// Mitsubishi GX Developer project: パレット移載装置   PLC: Q02

PROGRAM T-PANEL
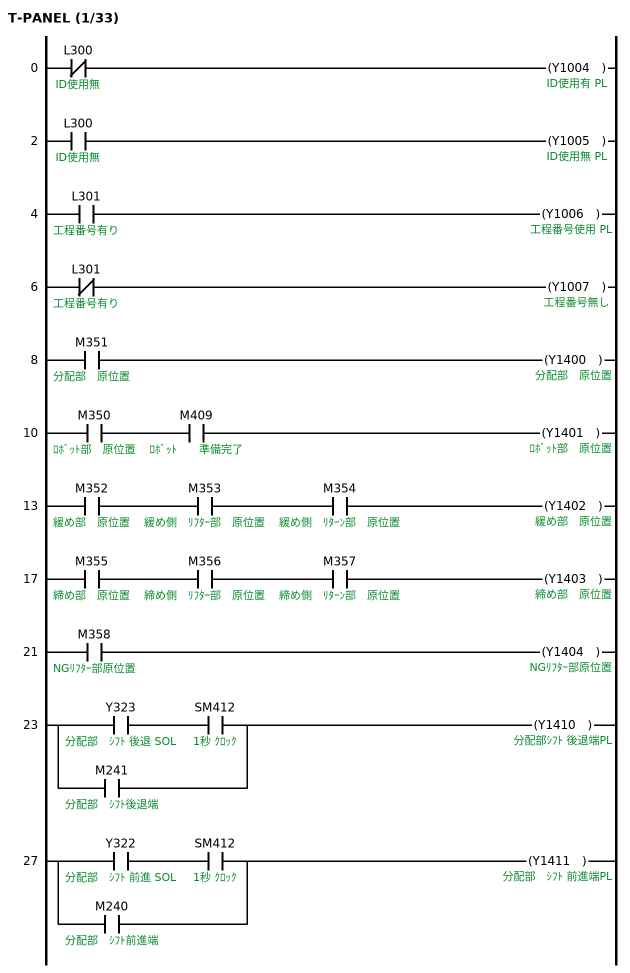
0     LDI     L300  ; ID使用無
      OUT     Y1004  ; ID使用有 PL
2     LD      L300  ; ID使用無
      OUT     Y1005  ; ID使用無 PL
4     LD      L301  ; 工程番号有り
      OUT     Y1006  ; 工程番号使用 PL
6     LDI     L301  ; 工程番号有り
      OUT     Y1007  ; 工程番号無し
8     LD      M351  ; 分配部　原位置
      OUT     Y1400  ; 分配部　原位置
10    LD      M350  ; ﾛﾎﾞｯﾄ部　原位置
      AND     M409  ; ﾛﾎﾞｯﾄ　　準備完了
      OUT     Y1401  ; ﾛﾎﾞｯﾄ部　原位置
13    LD      M352  ; 緩め部　原位置
      AND     M353  ; 緩め側　ﾘﾌﾀｰ部　原位置
      AND     M354  ; 緩め側　ﾘﾀｰﾝ部　原位置
      OUT     Y1402  ; 緩め部　原位置
17    LD      M355  ; 締め部　原位置
      AND     M356  ; 締め側　ﾘﾌﾀｰ部　原位置
      AND     M357  ; 締め側　ﾘﾀｰﾝ部　原位置
      OUT     Y1403  ; 締め部　原位置
21    LD      M358  ; NGﾘﾌﾀｰ部原位置
      OUT     Y1404  ; NGﾘﾌﾀｰ部原位置
23    LD      Y323  ; 分配部　ｼﾌﾄ 後退 SOL
      AND     SM412  ; 1秒 ｸﾛｯｸ
      OR      M241  ; 分配部　ｼﾌﾄ後退端
      OUT     Y1410  ; 分配部ｼﾌﾄ 後退端PL
27    LD      Y322  ; 分配部　ｼﾌﾄ 前進 SOL
      AND     SM412  ; 1秒 ｸﾛｯｸ
      OR      M240  ; 分配部　ｼﾌﾄ前進端
      OUT     Y1411  ; 分配部　ｼﾌﾄ 前進端PL
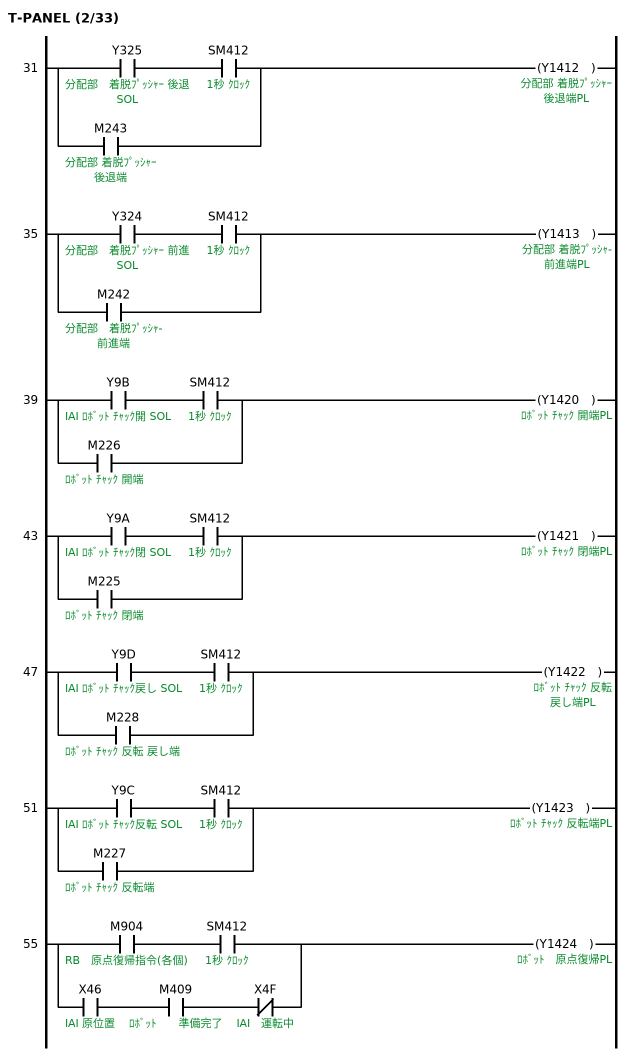
31    LD      Y325  ; 分配部　着脱ﾌﾟｯｼｬｰ 後退 SOL
      AND     SM412  ; 1秒 ｸﾛｯｸ
      OR      M243  ; 分配部 着脱ﾌﾟｯｼｬｰ 後退端
      OUT     Y1412  ; 分配部 着脱ﾌﾟｯｼｬｰ 後退端PL
35    LD      Y324  ; 分配部　着脱ﾌﾟｯｼｬｰ 前進 SOL
      AND     SM412  ; 1秒 ｸﾛｯｸ
      OR      M242  ; 分配部　着脱ﾌﾟｯｼｬ- 前進端
      OUT     Y1413  ; 分配部 着脱ﾌﾟｯｼｬ- 前進端PL
39    LD      Y9B  ; IAI ﾛﾎﾞｯﾄ ﾁｬｯｸ開 SOL
      AND     SM412  ; 1秒 ｸﾛｯｸ
      OR      M226  ; ﾛﾎﾞｯﾄ ﾁｬｯｸ 開端
      OUT     Y1420  ; ﾛﾎﾞｯﾄ ﾁｬｯｸ 開端PL
43    LD      Y9A  ; IAI ﾛﾎﾞｯﾄ ﾁｬｯｸ閉 SOL
      AND     SM412  ; 1秒 ｸﾛｯｸ
      OR      M225  ; ﾛﾎﾞｯﾄ ﾁｬｯｸ 閉端
      OUT     Y1421  ; ﾛﾎﾞｯﾄ ﾁｬｯｸ 閉端PL
47    LD      Y9D  ; IAI ﾛﾎﾞｯﾄ ﾁｬｯｸ戻し SOL
      AND     SM412  ; 1秒 ｸﾛｯｸ
      OR      M228  ; ﾛﾎﾞｯﾄ ﾁｬｯｸ 反転 戻し端
      OUT     Y1422  ; ﾛﾎﾞｯﾄ ﾁｬｯｸ 反転 戻し端PL
51    LD      Y9C  ; IAI ﾛﾎﾞｯﾄ ﾁｬｯｸ反転 SOL
      AND     SM412  ; 1秒 ｸﾛｯｸ
      OR      M227  ; ﾛﾎﾞｯﾄ ﾁｬｯｸ 反転端
      OUT     Y1423  ; ﾛﾎﾞｯﾄ ﾁｬｯｸ 反転端PL
55    LD      M904  ; RB　原点復帰指令(各個)
      AND     SM412  ; 1秒 ｸﾛｯｸ
      LD      X46  ; IAI 原位置
      AND     M409  ; ﾛﾎﾞｯﾄ　　準備完了
      ANI     X4F  ; IAI　運転中
      ORB
      OUT     Y1424  ; ﾛﾎﾞｯﾄ　原点復帰PL
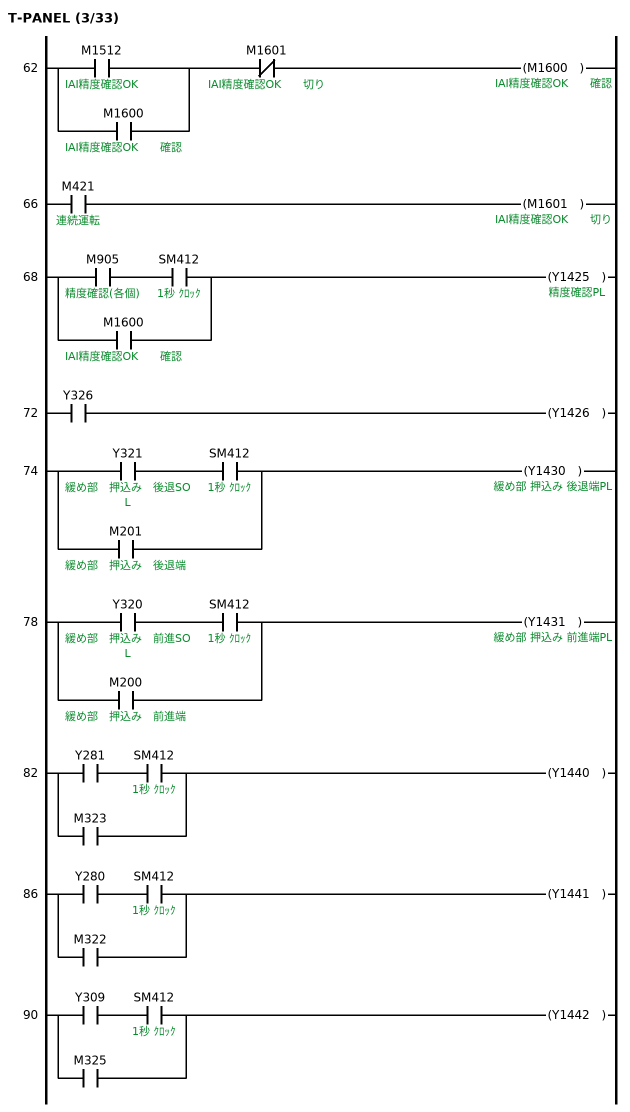
62    LD      M1512  ; IAI精度確認OK
      OR      M1600  ; IAI精度確認OK　　確認
      ANI     M1601  ; IAI精度確認OK　　切り
      OUT     M1600  ; IAI精度確認OK　　確認
66    LD      M421  ; 連続運転
      OUT     M1601  ; IAI精度確認OK　　切り
68    LD      M905  ; 精度確認(各個)
      AND     SM412  ; 1秒 ｸﾛｯｸ
      OR      M1600  ; IAI精度確認OK　　確認
      OUT     Y1425  ; 精度確認PL
72    LD      Y326
      OUT     Y1426
74    LD      Y321  ; 緩め部　押込み　後退SOL
      AND     SM412  ; 1秒 ｸﾛｯｸ
      OR      M201  ; 緩め部　押込み　後退端
      OUT     Y1430  ; 緩め部 押込み 後退端PL
78    LD      Y320  ; 緩め部　押込み　前進SOL
      AND     SM412  ; 1秒 ｸﾛｯｸ
      OR      M200  ; 緩め部　押込み　前進端
      OUT     Y1431  ; 緩め部 押込み 前進端PL
82    LD      Y281
      AND     SM412  ; 1秒 ｸﾛｯｸ
      OR      M323
      OUT     Y1440
86    LD      Y280
      AND     SM412  ; 1秒 ｸﾛｯｸ
      OR      M322
      OUT     Y1441
90    LD      Y309
      AND     SM412  ; 1秒 ｸﾛｯｸ
      OR      M325
      OUT     Y1442
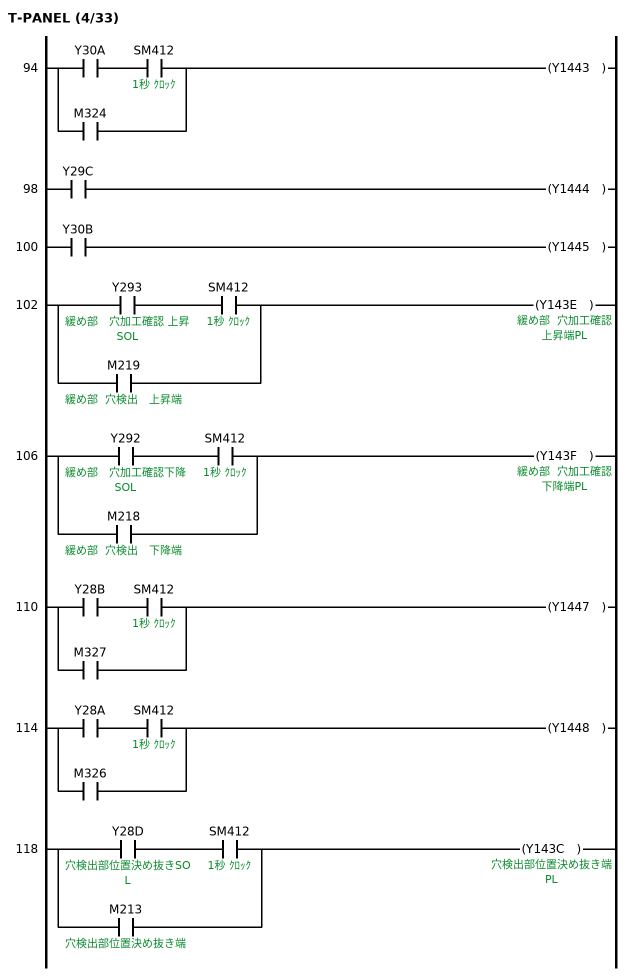
94    LD      Y30A
      AND     SM412  ; 1秒 ｸﾛｯｸ
      OR      M324
      OUT     Y1443
98    LD      Y29C
      OUT     Y1444
100   LD      Y30B
      OUT     Y1445
102   LD      Y293  ; 緩め部　穴加工確認 上昇 SOL
      AND     SM412  ; 1秒 ｸﾛｯｸ
      OR      M219  ; 緩め部  穴検出　上昇端
      OUT     Y143E  ; 緩め部  穴加工確認 上昇端PL
106   LD      Y292  ; 緩め部　穴加工確認下降 SOL
      AND     SM412  ; 1秒 ｸﾛｯｸ
      OR      M218  ; 緩め部  穴検出　下降端
      OUT     Y143F  ; 緩め部  穴加工確認 下降端PL
110   LD      Y28B
      AND     SM412  ; 1秒 ｸﾛｯｸ
      OR      M327
      OUT     Y1447
114   LD      Y28A
      AND     SM412  ; 1秒 ｸﾛｯｸ
      OR      M326
      OUT     Y1448
118   LD      Y28D  ; 穴検出部位置決め抜きSOL
      AND     SM412  ; 1秒 ｸﾛｯｸ
      OR      M213  ; 穴検出部位置決め抜き端
      OUT     Y143C  ; 穴検出部位置決め抜き端PL
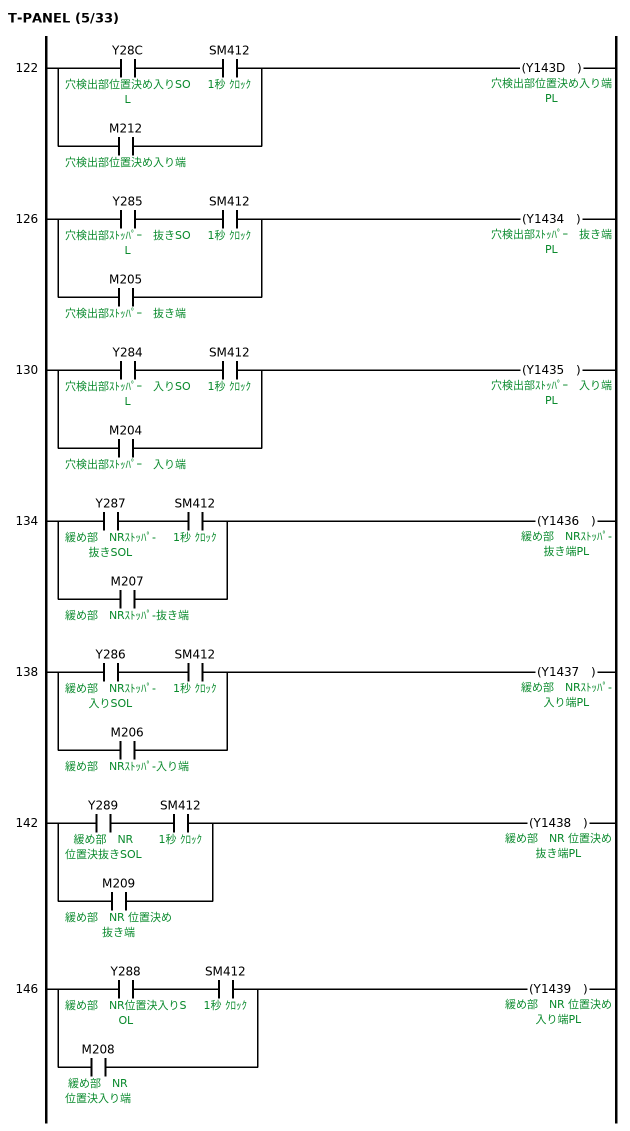
122   LD      Y28C  ; 穴検出部位置決め入りSOL
      AND     SM412  ; 1秒 ｸﾛｯｸ
      OR      M212  ; 穴検出部位置決め入り端
      OUT     Y143D  ; 穴検出部位置決め入り端PL
126   LD      Y285  ; 穴検出部ｽﾄｯﾊﾟｰ　抜きSOL
      AND     SM412  ; 1秒 ｸﾛｯｸ
      OR      M205  ; 穴検出部ｽﾄｯﾊﾟｰ　抜き端
      OUT     Y1434  ; 穴検出部ｽﾄｯﾊﾟｰ　抜き端PL
130   LD      Y284  ; 穴検出部ｽﾄｯﾊﾟｰ　入りSOL
      AND     SM412  ; 1秒 ｸﾛｯｸ
      OR      M204  ; 穴検出部ｽﾄｯﾊﾟｰ　入り端
      OUT     Y1435  ; 穴検出部ｽﾄｯﾊﾟｰ　入り端PL
134   LD      Y287  ; 緩め部　NRｽﾄｯﾊﾟ-抜きSOL
      AND     SM412  ; 1秒 ｸﾛｯｸ
      OR      M207  ; 緩め部　NRｽﾄｯﾊﾟ-抜き端
      OUT     Y1436  ; 緩め部　NRｽﾄｯﾊﾟ-抜き端PL
138   LD      Y286  ; 緩め部　NRｽﾄｯﾊﾟ-入りSOL
      AND     SM412  ; 1秒 ｸﾛｯｸ
      OR      M206  ; 緩め部　NRｽﾄｯﾊﾟ-入り端
      OUT     Y1437  ; 緩め部　NRｽﾄｯﾊﾟ-入り端PL
142   LD      Y289  ; 緩め部　NR 位置決抜きSOL
      AND     SM412  ; 1秒 ｸﾛｯｸ
      OR      M209  ; 緩め部　NR 位置決め 抜き端
      OUT     Y1438  ; 緩め部　NR 位置決め 抜き端PL
146   LD      Y288  ; 緩め部　NR位置決入りSOL
      AND     SM412  ; 1秒 ｸﾛｯｸ
      OR      M208  ; 緩め部　NR 位置決入り端
      OUT     Y1439  ; 緩め部　NR 位置決め 入り端PL
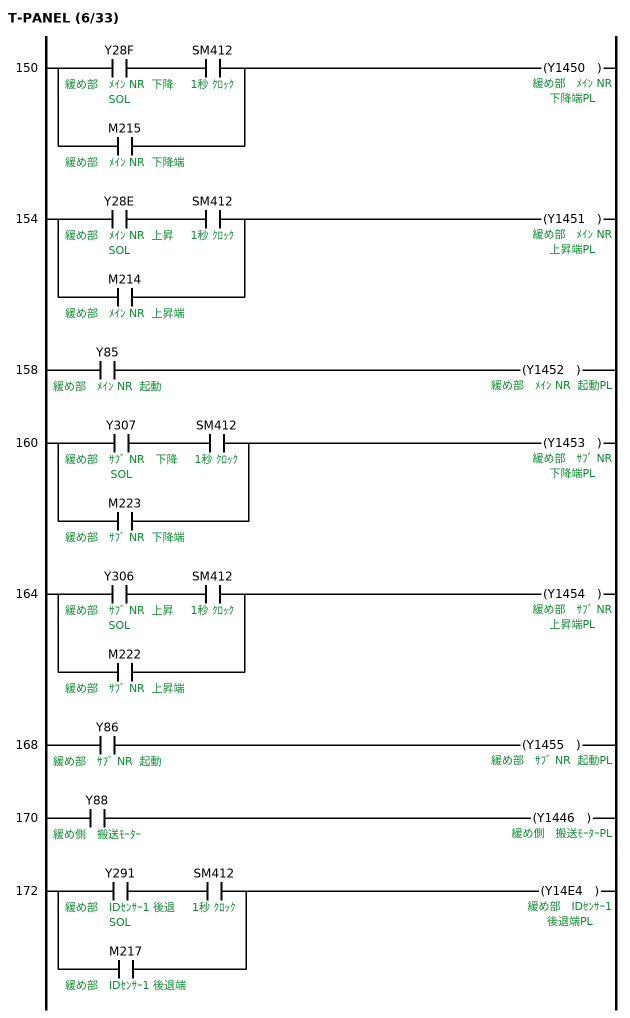
150   LD      Y28F  ; 緩め部　ﾒｲﾝ NR  下降 SOL
      AND     SM412  ; 1秒 ｸﾛｯｸ
      OR      M215  ; 緩め部　ﾒｲﾝ NR  下降端
      OUT     Y1450  ; 緩め部　ﾒｲﾝ NR  下降端PL
154   LD      Y28E  ; 緩め部　ﾒｲﾝ NR  上昇 SOL
      AND     SM412  ; 1秒 ｸﾛｯｸ
      OR      M214  ; 緩め部　ﾒｲﾝ NR  上昇端
      OUT     Y1451  ; 緩め部　ﾒｲﾝ NR  上昇端PL
158   LD      Y85  ; 緩め部　ﾒｲﾝ NR  起動
      OUT     Y1452  ; 緩め部　ﾒｲﾝ NR  起動PL
160   LD      Y307  ; 緩め部　ｻﾌﾞ NR　下降 SOL
      AND     SM412  ; 1秒 ｸﾛｯｸ
      OR      M223  ; 緩め部　ｻﾌﾞ NR  下降端
      OUT     Y1453  ; 緩め部　ｻﾌﾞ NR  下降端PL
164   LD      Y306  ; 緩め部　ｻﾌﾞ NR  上昇 SOL
      AND     SM412  ; 1秒 ｸﾛｯｸ
      OR      M222  ; 緩め部　ｻﾌﾞ NR  上昇端
      OUT     Y1454  ; 緩め部　ｻﾌﾞ NR  上昇端PL
168   LD      Y86  ; 緩め部　ｻﾌﾞ NR  起動
      OUT     Y1455  ; 緩め部　ｻﾌﾞ NR  起動PL
170   LD      Y88  ; 緩め側　搬送ﾓｰﾀｰ
      OUT     Y1446  ; 緩め側　搬送ﾓｰﾀｰPL
172   LD      Y291  ; 緩め部　IDｾﾝｻｰ1 後退 SOL
      AND     SM412  ; 1秒 ｸﾛｯｸ
      OR      M217  ; 緩め部　IDｾﾝｻｰ1 後退端
      OUT     Y14E4  ; 緩め部　IDｾﾝｻｰ1 後退端PL
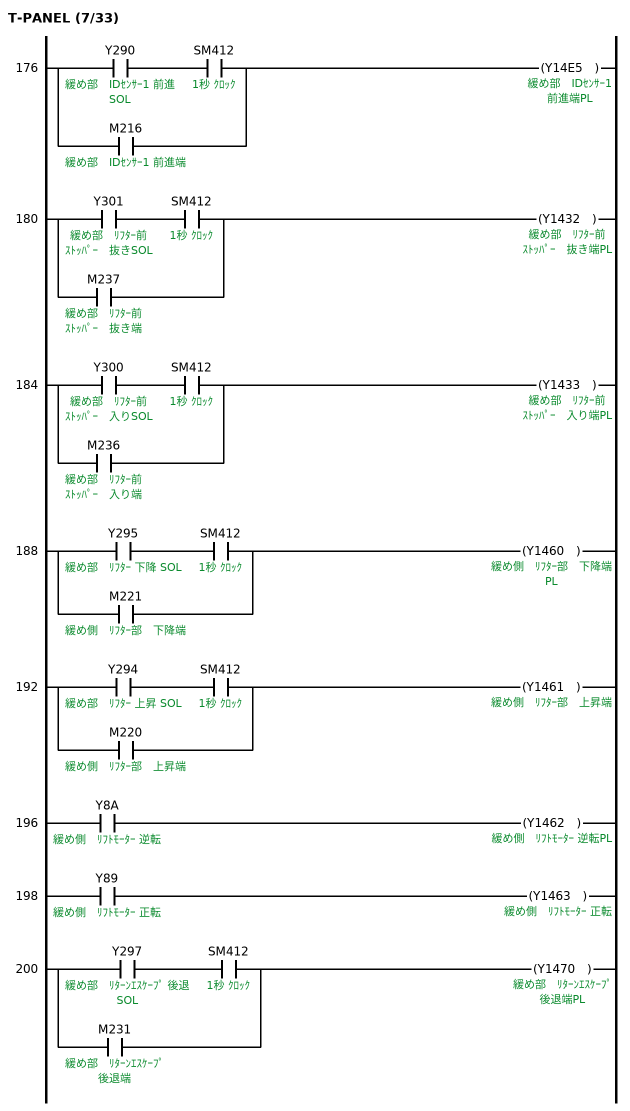
176   LD      Y290  ; 緩め部　IDｾﾝｻｰ1 前進 SOL
      AND     SM412  ; 1秒 ｸﾛｯｸ
      OR      M216  ; 緩め部　IDｾﾝｻｰ1 前進端
      OUT     Y14E5  ; 緩め部　IDｾﾝｻｰ1 前進端PL
180   LD      Y301  ; 緩め部　ﾘﾌﾀｰ前  ｽﾄｯﾊﾟｰ　抜きSOL
      AND     SM412  ; 1秒 ｸﾛｯｸ
      OR      M237  ; 緩め部　ﾘﾌﾀｰ前  ｽﾄｯﾊﾟｰ　抜き端
      OUT     Y1432  ; 緩め部　ﾘﾌﾀｰ前  ｽﾄｯﾊﾟｰ　抜き端PL
184   LD      Y300  ; 緩め部　ﾘﾌﾀｰ前  ｽﾄｯﾊﾟｰ　入りSOL
      AND     SM412  ; 1秒 ｸﾛｯｸ
      OR      M236  ; 緩め部　ﾘﾌﾀｰ前  ｽﾄｯﾊﾟｰ　入り端
      OUT     Y1433  ; 緩め部　ﾘﾌﾀｰ前  ｽﾄｯﾊﾟｰ　入り端PL
188   LD      Y295  ; 緩め部　ﾘﾌﾀｰ 下降 SOL
      AND     SM412  ; 1秒 ｸﾛｯｸ
      OR      M221  ; 緩め側　ﾘﾌﾀｰ部　下降端
      OUT     Y1460  ; 緩め側　ﾘﾌﾀｰ部　下降端PL
192   LD      Y294  ; 緩め部　ﾘﾌﾀｰ 上昇 SOL
      AND     SM412  ; 1秒 ｸﾛｯｸ
      OR      M220  ; 緩め側　ﾘﾌﾀｰ部　上昇端
      OUT     Y1461  ; 緩め側　ﾘﾌﾀｰ部　上昇端
196   LD      Y8A  ; 緩め側　ﾘﾌﾄﾓｰﾀｰ 逆転
      OUT     Y1462  ; 緩め側　ﾘﾌﾄﾓｰﾀｰ 逆転PL
198   LD      Y89  ; 緩め側　ﾘﾌﾄﾓｰﾀｰ 正転
      OUT     Y1463  ; 緩め側　ﾘﾌﾄﾓｰﾀｰ 正転
200   LD      Y297  ; 緩め部　ﾘﾀｰﾝｴｽｹｰﾌﾟ 後退 SOL
      AND     SM412  ; 1秒 ｸﾛｯｸ
      OR      M231  ; 緩め部　ﾘﾀｰﾝｴｽｹｰﾌﾟ 後退端
      OUT     Y1470  ; 緩め部　ﾘﾀｰﾝｴｽｹｰﾌﾟ 後退端PL
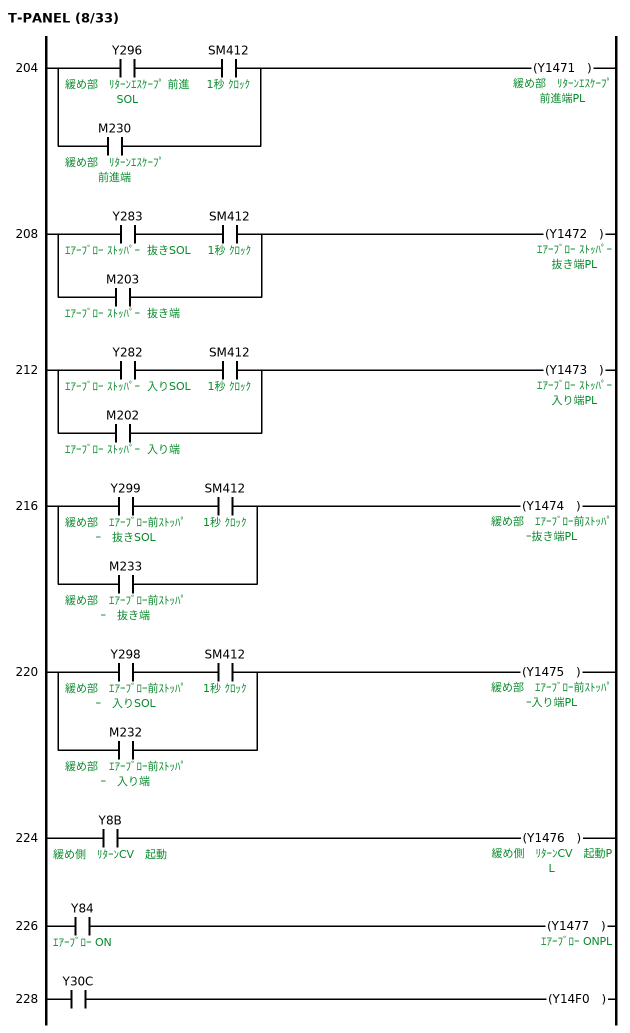
204   LD      Y296  ; 緩め部　ﾘﾀｰﾝｴｽｹｰﾌﾟ 前進 SOL
      AND     SM412  ; 1秒 ｸﾛｯｸ
      OR      M230  ; 緩め部　ﾘﾀｰﾝｴｽｹｰﾌﾟ 前進端
      OUT     Y1471  ; 緩め部　ﾘﾀｰﾝｴｽｹｰﾌﾟ 前進端PL
208   LD      Y283  ; ｴｱｰﾌﾞﾛｰ ｽﾄｯﾊﾟｰ  抜きSOL
      AND     SM412  ; 1秒 ｸﾛｯｸ
      OR      M203  ; ｴｱｰﾌﾞﾛｰ ｽﾄｯﾊﾟｰ  抜き端
      OUT     Y1472  ; ｴｱｰﾌﾞﾛｰ ｽﾄｯﾊﾟｰ  抜き端PL
212   LD      Y282  ; ｴｱｰﾌﾞﾛｰ ｽﾄｯﾊﾟｰ  入りSOL
      AND     SM412  ; 1秒 ｸﾛｯｸ
      OR      M202  ; ｴｱｰﾌﾞﾛｰ ｽﾄｯﾊﾟｰ  入り端
      OUT     Y1473  ; ｴｱｰﾌﾞﾛｰ ｽﾄｯﾊﾟｰ  入り端PL
216   LD      Y299  ; 緩め部　ｴｱｰﾌﾞﾛｰ前ｽﾄｯﾊﾟｰ　抜きSOL
      AND     SM412  ; 1秒 ｸﾛｯｸ
      OR      M233  ; 緩め部　ｴｱｰﾌﾞﾛｰ前ｽﾄｯﾊﾟｰ　抜き端
      OUT     Y1474  ; 緩め部　ｴｱｰﾌﾞﾛｰ前ｽﾄｯﾊﾟｰ抜き端PL
220   LD      Y298  ; 緩め部　ｴｱｰﾌﾞﾛｰ前ｽﾄｯﾊﾟｰ　入りSOL
      AND     SM412  ; 1秒 ｸﾛｯｸ
      OR      M232  ; 緩め部　ｴｱｰﾌﾞﾛｰ前ｽﾄｯﾊﾟｰ　入り端
      OUT     Y1475  ; 緩め部　ｴｱｰﾌﾞﾛｰ前ｽﾄｯﾊﾟｰ入り端PL
224   LD      Y8B  ; 緩め側　ﾘﾀｰﾝCV　起動
      OUT     Y1476  ; 緩め側　ﾘﾀｰﾝCV　起動PL
226   LD      Y84  ; ｴｱｰﾌﾞﾛｰ ON
      OUT     Y1477  ; ｴｱｰﾌﾞﾛｰ ONPL
228   LD      Y30C
      OUT     Y14F0
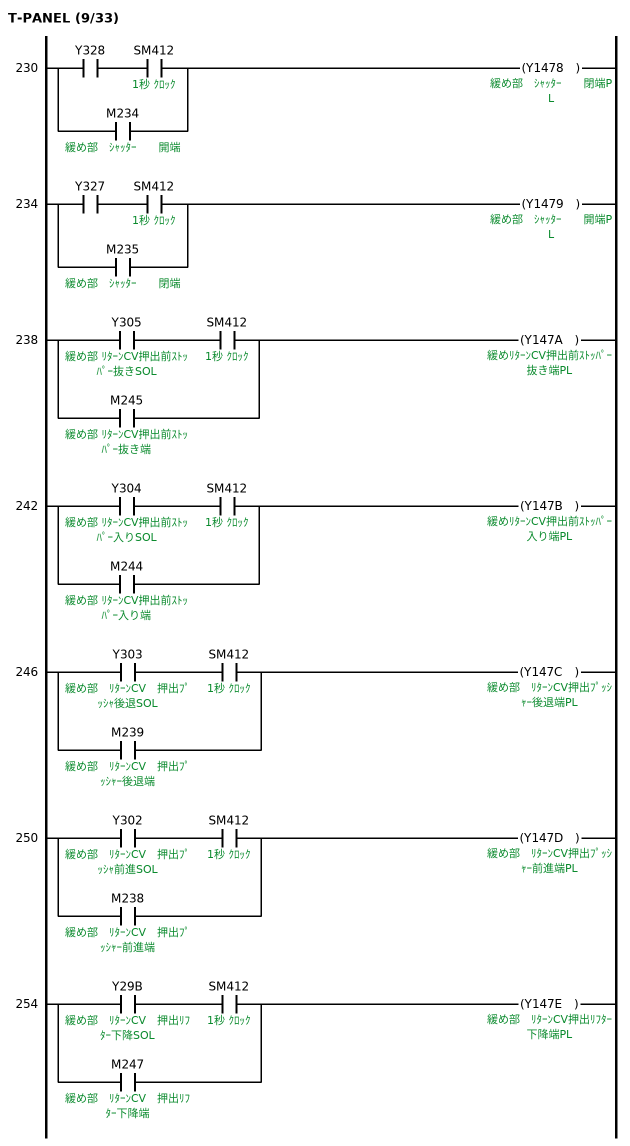
230   LD      Y328
      AND     SM412  ; 1秒 ｸﾛｯｸ
      OR      M234  ; 緩め部　ｼｬｯﾀｰ　　開端
      OUT     Y1478  ; 緩め部　ｼｬｯﾀｰ　　閉端PL
234   LD      Y327
      AND     SM412  ; 1秒 ｸﾛｯｸ
      OR      M235  ; 緩め部　ｼｬｯﾀｰ　　閉端
      OUT     Y1479  ; 緩め部　ｼｬｯﾀｰ　　開端PL
238   LD      Y305  ; 緩め部 ﾘﾀｰﾝCV押出前ｽﾄｯﾊﾟｰ抜きSOL
      AND     SM412  ; 1秒 ｸﾛｯｸ
      OR      M245  ; 緩め部 ﾘﾀｰﾝCV押出前ｽﾄｯﾊﾟｰ抜き端
      OUT     Y147A  ; 緩めﾘﾀｰﾝCV押出前ｽﾄｯﾊﾟｰ抜き端PL
242   LD      Y304  ; 緩め部 ﾘﾀｰﾝCV押出前ｽﾄｯﾊﾟｰ入りSOL
      AND     SM412  ; 1秒 ｸﾛｯｸ
      OR      M244  ; 緩め部 ﾘﾀｰﾝCV押出前ｽﾄｯﾊﾟｰ入り端
      OUT     Y147B  ; 緩めﾘﾀｰﾝCV押出前ｽﾄｯﾊﾟｰ入り端PL
246   LD      Y303  ; 緩め部　ﾘﾀｰﾝCV　押出ﾌﾟｯｼｬ後退SOL
      AND     SM412  ; 1秒 ｸﾛｯｸ
      OR      M239  ; 緩め部　ﾘﾀｰﾝCV　押出ﾌﾟｯｼｬｰ後退端
      OUT     Y147C  ; 緩め部　ﾘﾀｰﾝCV押出ﾌﾟｯｼｬｰ後退端PL
250   LD      Y302  ; 緩め部　ﾘﾀｰﾝCV　押出ﾌﾟｯｼｬ前進SOL
      AND     SM412  ; 1秒 ｸﾛｯｸ
      OR      M238  ; 緩め部　ﾘﾀｰﾝCV　押出ﾌﾟｯｼｬｰ前進端
      OUT     Y147D  ; 緩め部　ﾘﾀｰﾝCV押出ﾌﾟｯｼｬｰ前進端PL
254   LD      Y29B  ; 緩め部　ﾘﾀｰﾝCV　押出ﾘﾌﾀｰ下降SOL
      AND     SM412  ; 1秒 ｸﾛｯｸ
      OR      M247  ; 緩め部　ﾘﾀｰﾝCV　押出ﾘﾌﾀｰ下降端
      OUT     Y147E  ; 緩め部　ﾘﾀｰﾝCV押出ﾘﾌﾀｰ下降端PL
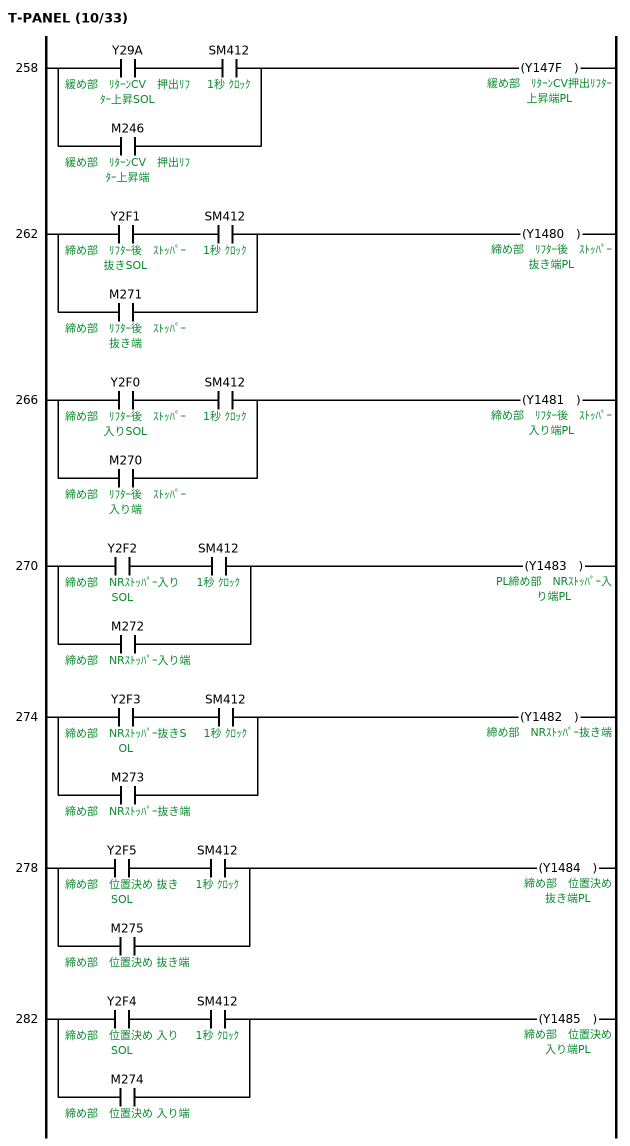
258   LD      Y29A  ; 緩め部　ﾘﾀｰﾝCV　押出ﾘﾌﾀｰ上昇SOL
      AND     SM412  ; 1秒 ｸﾛｯｸ
      OR      M246  ; 緩め部　ﾘﾀｰﾝCV　押出ﾘﾌﾀｰ上昇端
      OUT     Y147F  ; 緩め部　ﾘﾀｰﾝCV押出ﾘﾌﾀｰ上昇端PL
262   LD      Y2F1  ; 締め部　ﾘﾌﾀｰ後　ｽﾄｯﾊﾟｰ　抜きSOL
      AND     SM412  ; 1秒 ｸﾛｯｸ
      OR      M271  ; 締め部　ﾘﾌﾀｰ後　ｽﾄｯﾊﾟｰ　抜き端
      OUT     Y1480  ; 締め部　ﾘﾌﾀｰ後　ｽﾄｯﾊﾟｰ　抜き端PL
266   LD      Y2F0  ; 締め部　ﾘﾌﾀｰ後　ｽﾄｯﾊﾟｰ　入りSOL
      AND     SM412  ; 1秒 ｸﾛｯｸ
      OR      M270  ; 締め部　ﾘﾌﾀｰ後　ｽﾄｯﾊﾟｰ　入り端
      OUT     Y1481  ; 締め部　ﾘﾌﾀｰ後　ｽﾄｯﾊﾟｰ　入り端PL
270   LD      Y2F2  ; 締め部　NRｽﾄｯﾊﾟｰ入り SOL
      AND     SM412  ; 1秒 ｸﾛｯｸ
      OR      M272  ; 締め部　NRｽﾄｯﾊﾟｰ入り端
      OUT     Y1483  ; PL締め部　NRｽﾄｯﾊﾟｰ入り端PL
274   LD      Y2F3  ; 締め部　NRｽﾄｯﾊﾟｰ抜きSOL
      AND     SM412  ; 1秒 ｸﾛｯｸ
      OR      M273  ; 締め部　NRｽﾄｯﾊﾟｰ抜き端
      OUT     Y1482  ; 締め部　NRｽﾄｯﾊﾟｰ抜き端
278   LD      Y2F5  ; 締め部　位置決め 抜き SOL
      AND     SM412  ; 1秒 ｸﾛｯｸ
      OR      M275  ; 締め部　位置決め 抜き端
      OUT     Y1484  ; 締め部　位置決め 抜き端PL
282   LD      Y2F4  ; 締め部　位置決め 入り SOL
      AND     SM412  ; 1秒 ｸﾛｯｸ
      OR      M274  ; 締め部　位置決め 入り端
      OUT     Y1485  ; 締め部　位置決め 入り端PL
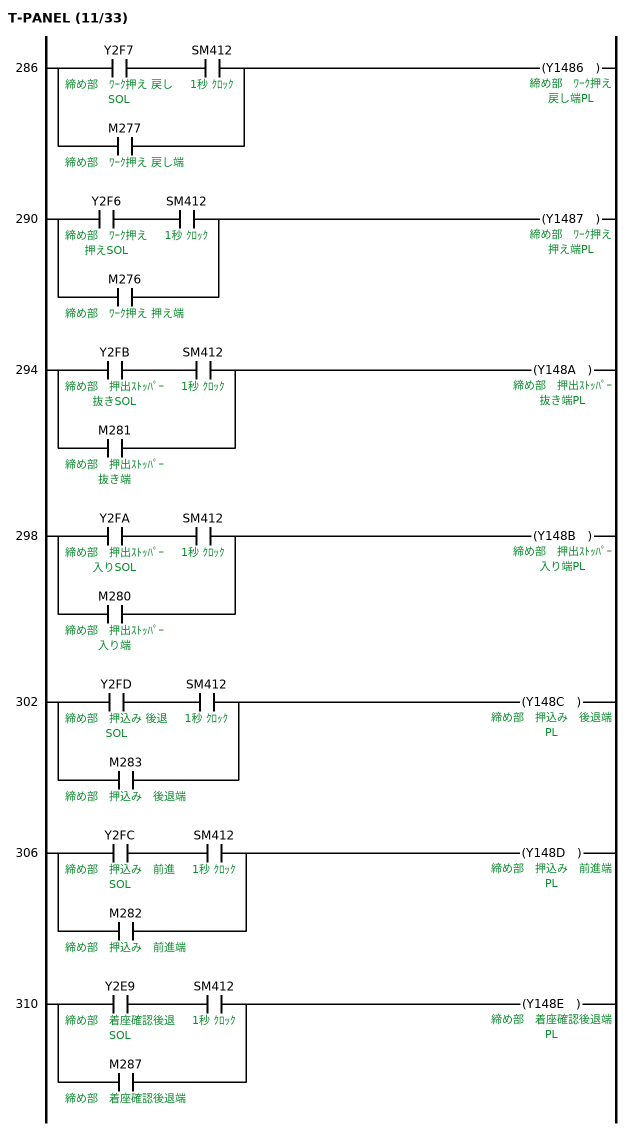
286   LD      Y2F7  ; 締め部　ﾜｰｸ押え 戻し SOL
      AND     SM412  ; 1秒 ｸﾛｯｸ
      OR      M277  ; 締め部　ﾜｰｸ押え 戻し端
      OUT     Y1486  ; 締め部　ﾜｰｸ押え 戻し端PL
290   LD      Y2F6  ; 締め部　ﾜｰｸ押え 押えSOL
      AND     SM412  ; 1秒 ｸﾛｯｸ
      OR      M276  ; 締め部　ﾜｰｸ押え 押え端
      OUT     Y1487  ; 締め部　ﾜｰｸ押え 押え端PL
294   LD      Y2FB  ; 締め部　押出ｽﾄｯﾊﾟｰ 抜きSOL
      AND     SM412  ; 1秒 ｸﾛｯｸ
      OR      M281  ; 締め部　押出ｽﾄｯﾊﾟｰ 抜き端
      OUT     Y148A  ; 締め部　押出ｽﾄｯﾊﾟｰ 抜き端PL
298   LD      Y2FA  ; 締め部　押出ｽﾄｯﾊﾟｰ 入りSOL
      AND     SM412  ; 1秒 ｸﾛｯｸ
      OR      M280  ; 締め部　押出ｽﾄｯﾊﾟｰ 入り端
      OUT     Y148B  ; 締め部　押出ｽﾄｯﾊﾟｰ 入り端PL
302   LD      Y2FD  ; 締め部　押込み 後退 SOL
      AND     SM412  ; 1秒 ｸﾛｯｸ
      OR      M283  ; 締め部　押込み　後退端
      OUT     Y148C  ; 締め部　押込み　後退端PL
306   LD      Y2FC  ; 締め部　押込み　前進 SOL
      AND     SM412  ; 1秒 ｸﾛｯｸ
      OR      M282  ; 締め部　押込み　前進端
      OUT     Y148D  ; 締め部　押込み　前進端PL
310   LD      Y2E9  ; 締め部　着座確認後退 SOL
      AND     SM412  ; 1秒 ｸﾛｯｸ
      OR      M287  ; 締め部　着座確認後退端
      OUT     Y148E  ; 締め部　着座確認後退端PL
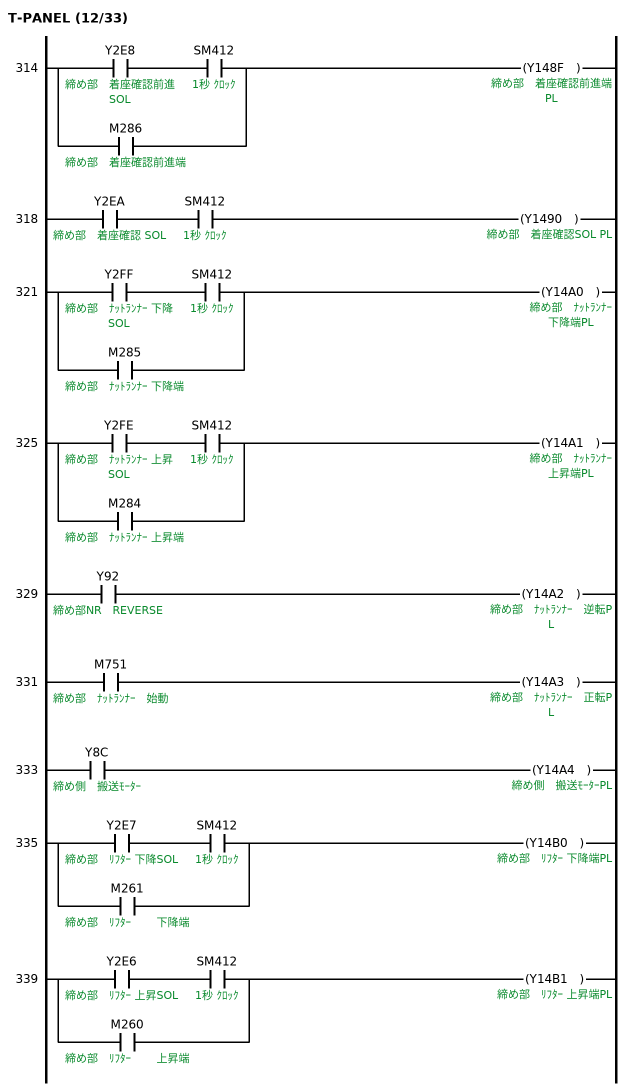
314   LD      Y2E8  ; 締め部　着座確認前進 SOL
      AND     SM412  ; 1秒 ｸﾛｯｸ
      OR      M286  ; 締め部　着座確認前進端
      OUT     Y148F  ; 締め部　着座確認前進端PL
318   LD      Y2EA  ; 締め部　着座確認 SOL
      AND     SM412  ; 1秒 ｸﾛｯｸ
      OUT     Y1490  ; 締め部　着座確認SOL PL
321   LD      Y2FF  ; 締め部　ﾅｯﾄﾗﾝﾅｰ 下降 SOL
      AND     SM412  ; 1秒 ｸﾛｯｸ
      OR      M285  ; 締め部　ﾅｯﾄﾗﾝﾅｰ 下降端
      OUT     Y14A0  ; 締め部　ﾅｯﾄﾗﾝﾅｰ 下降端PL
325   LD      Y2FE  ; 締め部　ﾅｯﾄﾗﾝﾅｰ 上昇 SOL
      AND     SM412  ; 1秒 ｸﾛｯｸ
      OR      M284  ; 締め部　ﾅｯﾄﾗﾝﾅｰ 上昇端
      OUT     Y14A1  ; 締め部　ﾅｯﾄﾗﾝﾅｰ 上昇端PL
329   LD      Y92  ; 締め部NR　REVERSE
      OUT     Y14A2  ; 締め部　ﾅｯﾄﾗﾝﾅｰ　逆転PL
331   LD      M751  ; 締め部　ﾅｯﾄﾗﾝﾅｰ　始動
      OUT     Y14A3  ; 締め部　ﾅｯﾄﾗﾝﾅｰ　正転PL
333   LD      Y8C  ; 締め側　搬送ﾓｰﾀｰ
      OUT     Y14A4  ; 締め側　搬送ﾓｰﾀｰPL
335   LD      Y2E7  ; 締め部　ﾘﾌﾀｰ 下降SOL
      AND     SM412  ; 1秒 ｸﾛｯｸ
      OR      M261  ; 締め部　ﾘﾌﾀｰ 　　下降端
      OUT     Y14B0  ; 締め部　ﾘﾌﾀｰ 下降端PL
339   LD      Y2E6  ; 締め部　ﾘﾌﾀｰ 上昇SOL
      AND     SM412  ; 1秒 ｸﾛｯｸ
      OR      M260  ; 締め部　ﾘﾌﾀｰ 　　上昇端
      OUT     Y14B1  ; 締め部　ﾘﾌﾀｰ 上昇端PL
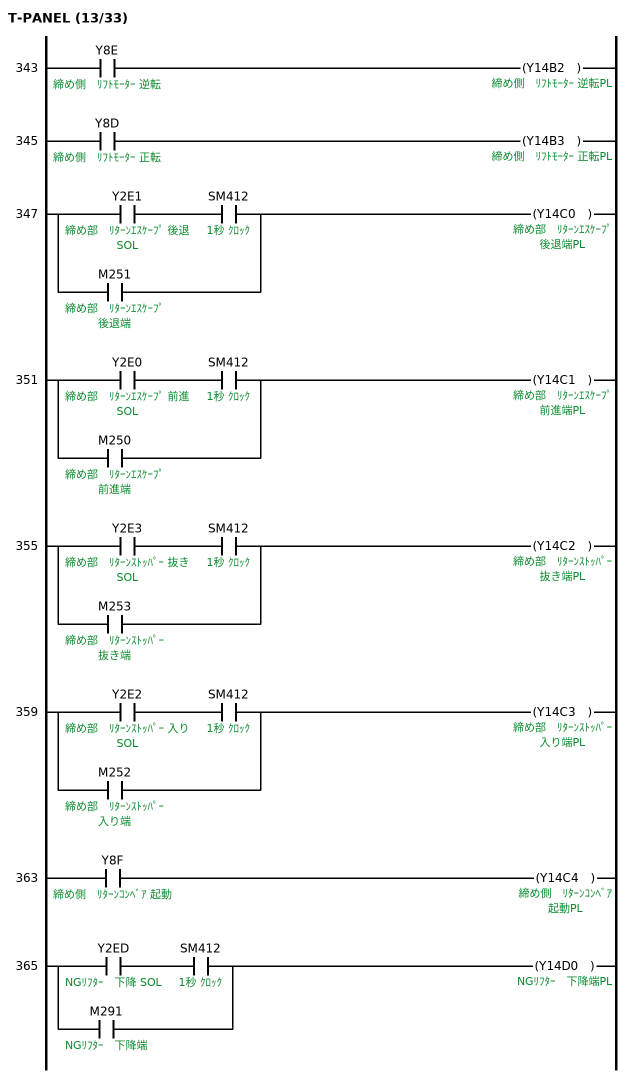
343   LD      Y8E  ; 締め側　ﾘﾌﾄﾓｰﾀｰ 逆転
      OUT     Y14B2  ; 締め側　ﾘﾌﾄﾓｰﾀｰ 逆転PL
345   LD      Y8D  ; 締め側　ﾘﾌﾄﾓｰﾀｰ 正転
      OUT     Y14B3  ; 締め側　ﾘﾌﾄﾓｰﾀｰ 正転PL
347   LD      Y2E1  ; 締め部　ﾘﾀｰﾝｴｽｹｰﾌﾟ 後退 SOL
      AND     SM412  ; 1秒 ｸﾛｯｸ
      OR      M251  ; 締め部　ﾘﾀｰﾝｴｽｹｰﾌﾟ 後退端
      OUT     Y14C0  ; 締め部　ﾘﾀｰﾝｴｽｹｰﾌﾟ 後退端PL
351   LD      Y2E0  ; 締め部　ﾘﾀｰﾝｴｽｹｰﾌﾟ 前進 SOL
      AND     SM412  ; 1秒 ｸﾛｯｸ
      OR      M250  ; 締め部　ﾘﾀｰﾝｴｽｹｰﾌﾟ 前進端
      OUT     Y14C1  ; 締め部　ﾘﾀｰﾝｴｽｹｰﾌﾟ 前進端PL
355   LD      Y2E3  ; 締め部　ﾘﾀｰﾝｽﾄｯﾊﾟｰ 抜き SOL
      AND     SM412  ; 1秒 ｸﾛｯｸ
      OR      M253  ; 締め部　ﾘﾀｰﾝｽﾄｯﾊﾟｰ 抜き端
      OUT     Y14C2  ; 締め部　ﾘﾀｰﾝｽﾄｯﾊﾟｰ 抜き端PL
359   LD      Y2E2  ; 締め部　ﾘﾀｰﾝｽﾄｯﾊﾟｰ 入り SOL
      AND     SM412  ; 1秒 ｸﾛｯｸ
      OR      M252  ; 締め部　ﾘﾀｰﾝｽﾄｯﾊﾟｰ 入り端
      OUT     Y14C3  ; 締め部　ﾘﾀｰﾝｽﾄｯﾊﾟｰ 入り端PL
363   LD      Y8F  ; 締め側　ﾘﾀｰﾝｺﾝﾍﾞｱ 起動
      OUT     Y14C4  ; 締め側　ﾘﾀｰﾝｺﾝﾍﾞｱ 起動PL
365   LD      Y2ED  ; NGﾘﾌﾀｰ　下降 SOL
      AND     SM412  ; 1秒 ｸﾛｯｸ
      OR      M291  ; NGﾘﾌﾀｰ　下降端
      OUT     Y14D0  ; NGﾘﾌﾀｰ　下降端PL
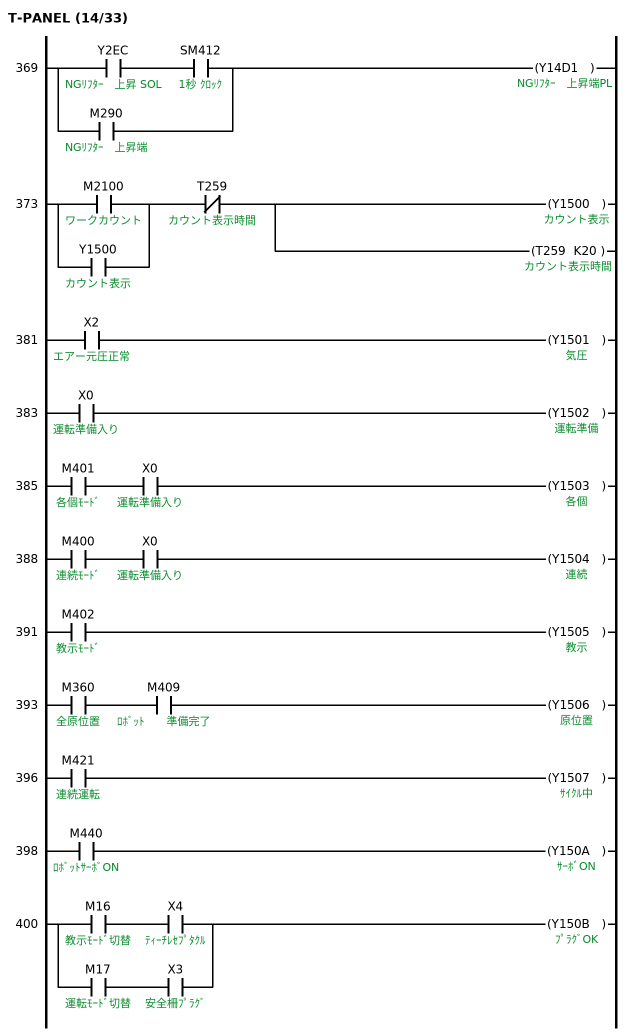
369   LD      Y2EC  ; NGﾘﾌﾀｰ　上昇 SOL
      AND     SM412  ; 1秒 ｸﾛｯｸ
      OR      M290  ; NGﾘﾌﾀｰ　上昇端
      OUT     Y14D1  ; NGﾘﾌﾀｰ　上昇端PL
373   LD      M2100  ; ワークカウント
      OR      Y1500  ; カウント表示
      ANI     T259  ; カウント表示時間
      OUT     Y1500  ; カウント表示
      OUT     T259 K20  ; カウント表示時間
381   LD      X2  ; エアー元圧正常
      OUT     Y1501  ; 気圧
383   LD      X0  ; 運転準備入り
      OUT     Y1502  ; 運転準備
385   LD      M401  ; 各個ﾓｰﾄﾞ
      AND     X0  ; 運転準備入り
      OUT     Y1503  ; 各個
388   LD      M400  ; 連続ﾓｰﾄﾞ
      AND     X0  ; 運転準備入り
      OUT     Y1504  ; 連続
391   LD      M402  ; 教示ﾓｰﾄﾞ
      OUT     Y1505  ; 教示
393   LD      M360  ; 全原位置
      AND     M409  ; ﾛﾎﾞｯﾄ　　準備完了
      OUT     Y1506  ; 原位置
396   LD      M421  ; 連続運転
      OUT     Y1507  ; ｻｲｸﾙ中
398   LD      M440  ; ﾛﾎﾞｯﾄｻｰﾎﾞON
      OUT     Y150A  ; ｻｰﾎﾞON
400   LD      M16  ; 教示ﾓｰﾄﾞ切替
      AND     X4  ; ﾃｨｰﾁﾚｾﾌﾟﾀｸﾙ
      LD      M17  ; 運転ﾓｰﾄﾞ切替
      AND     X3  ; 安全柵ﾌﾟﾗｸﾞ
      ORB
      OUT     Y150B  ; ﾌﾟﾗｸﾞOK
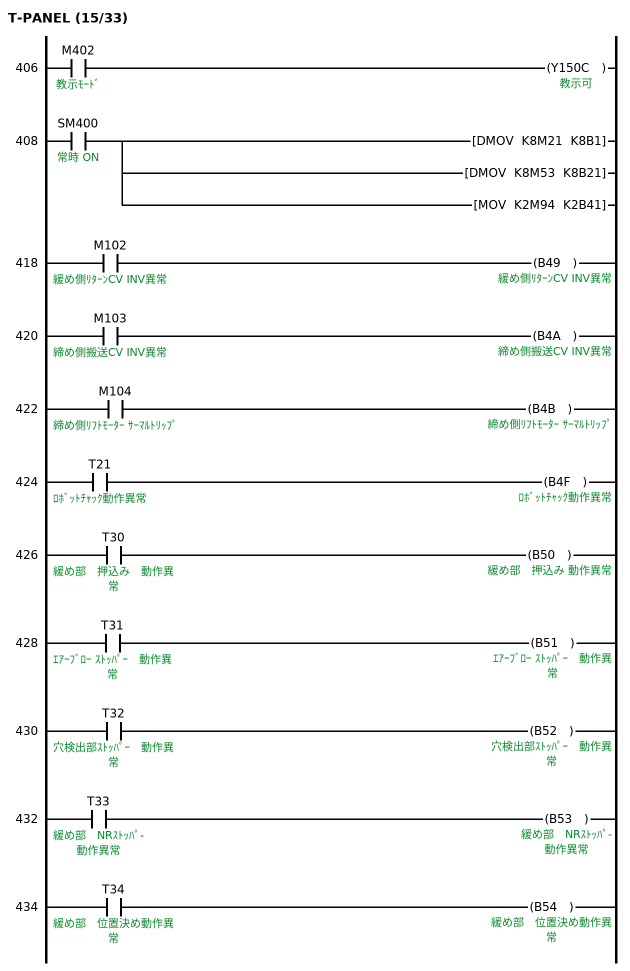
406   LD      M402  ; 教示ﾓｰﾄﾞ
      OUT     Y150C  ; 教示可
408   LD      SM400  ; 常時 ON
      DMOV    K8M21 K8B1  ; PC電池異常 / PC電池異常
      DMOV    K8M53 K8B21  ; 予備 / 予備
      MOV     K2M94 K2B41  ; ﾊﾟﾚｯﾄID異常 / ﾊﾟﾚｯﾄID異常
418   LD      M102  ; 緩め側ﾘﾀｰﾝCV INV異常
      OUT     B49  ; 緩め側ﾘﾀｰﾝCV INV異常
420   LD      M103  ; 締め側搬送CV INV異常
      OUT     B4A  ; 締め側搬送CV INV異常
422   LD      M104  ; 締め側ﾘﾌﾄﾓｰﾀｰ ｻｰﾏﾙﾄﾘｯﾌﾟ
      OUT     B4B  ; 締め側ﾘﾌﾄﾓｰﾀｰ ｻｰﾏﾙﾄﾘｯﾌﾟ
424   LD      T21  ; ﾛﾎﾞｯﾄﾁｬｯｸ動作異常
      OUT     B4F  ; ﾛﾎﾞｯﾄﾁｬｯｸ動作異常
426   LD      T30  ; 緩め部　押込み　動作異常
      OUT     B50  ; 緩め部　押込み 動作異常
428   LD      T31  ; ｴｱｰﾌﾞﾛｰ ｽﾄｯﾊﾟｰ　動作異常
      OUT     B51  ; ｴｱｰﾌﾞﾛｰ ｽﾄｯﾊﾟｰ　動作異常
430   LD      T32  ; 穴検出部ｽﾄｯﾊﾟｰ　動作異常
      OUT     B52  ; 穴検出部ｽﾄｯﾊﾟｰ　動作異常
432   LD      T33  ; 緩め部　NRｽﾄｯﾊﾟ-動作異常
      OUT     B53  ; 緩め部　NRｽﾄｯﾊﾟ-動作異常
434   LD      T34  ; 緩め部　位置決め動作異常
      OUT     B54  ; 緩め部　位置決め動作異常
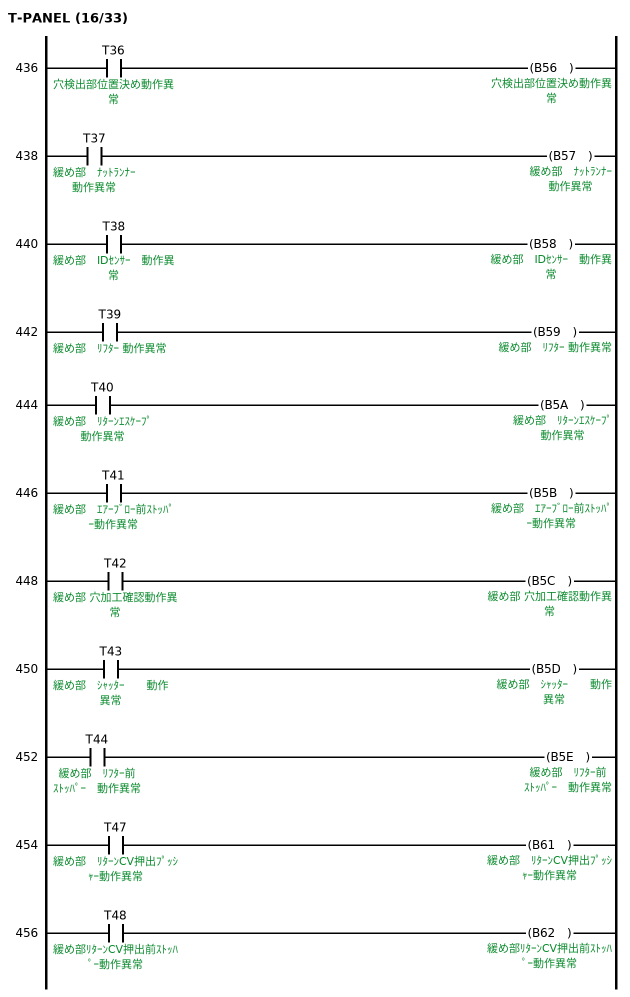
436   LD      T36  ; 穴検出部位置決め動作異常
      OUT     B56  ; 穴検出部位置決め動作異常
438   LD      T37  ; 緩め部　ﾅｯﾄﾗﾝﾅｰ 動作異常
      OUT     B57  ; 緩め部　ﾅｯﾄﾗﾝﾅｰ 動作異常
440   LD      T38  ; 緩め部　IDｾﾝｻｰ　動作異常
      OUT     B58  ; 緩め部　IDｾﾝｻｰ　動作異常
442   LD      T39  ; 緩め部　ﾘﾌﾀｰ 動作異常
      OUT     B59  ; 緩め部　ﾘﾌﾀｰ 動作異常
444   LD      T40  ; 緩め部　ﾘﾀｰﾝｴｽｹｰﾌﾟ 動作異常
      OUT     B5A  ; 緩め部　ﾘﾀｰﾝｴｽｹｰﾌﾟ 動作異常
446   LD      T41  ; 緩め部　ｴｱｰﾌﾞﾛｰ前ｽﾄｯﾊﾟｰ動作異常
      OUT     B5B  ; 緩め部　ｴｱｰﾌﾞﾛｰ前ｽﾄｯﾊﾟｰ動作異常
448   LD      T42  ; 緩め部 穴加工確認動作異常
      OUT     B5C  ; 緩め部 穴加工確認動作異常
450   LD      T43  ; 緩め部　ｼｬｯﾀｰ　　動作異常
      OUT     B5D  ; 緩め部　ｼｬｯﾀｰ　　動作異常
452   LD      T44  ; 緩め部　ﾘﾌﾀｰ前  ｽﾄｯﾊﾟｰ　動作異常
      OUT     B5E  ; 緩め部　ﾘﾌﾀｰ前  ｽﾄｯﾊﾟｰ　動作異常
454   LD      T47  ; 緩め部　ﾘﾀｰﾝCV押出ﾌﾟｯｼｬｰ動作異常
      OUT     B61  ; 緩め部　ﾘﾀｰﾝCV押出ﾌﾟｯｼｬｰ動作異常
456   LD      T48  ; 緩め部ﾘﾀｰﾝCV押出前ｽﾄｯﾊﾟｰ動作異常
      OUT     B62  ; 緩め部ﾘﾀｰﾝCV押出前ｽﾄｯﾊﾟｰ動作異常
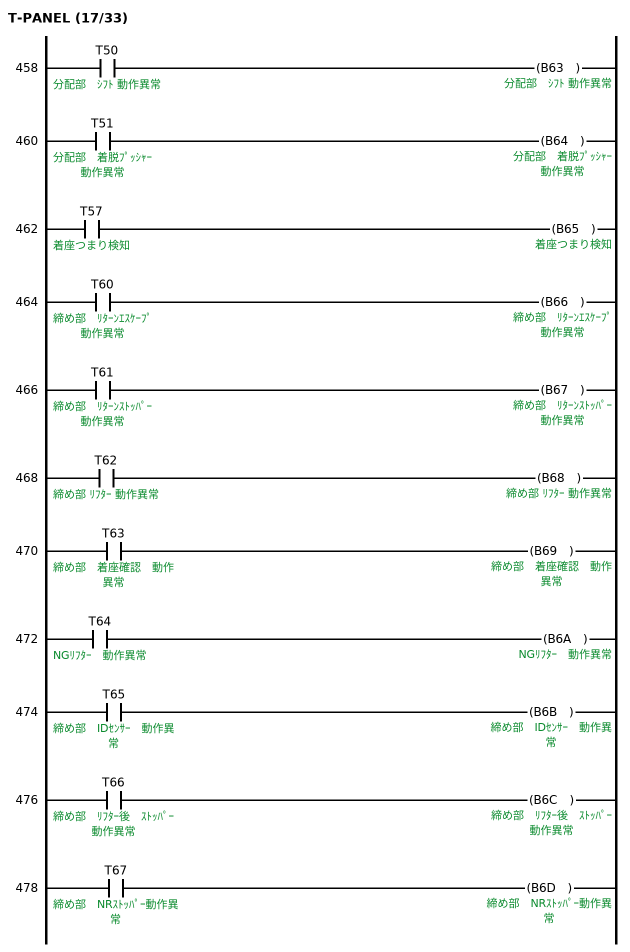
458   LD      T50  ; 分配部　ｼﾌﾄ 動作異常
      OUT     B63  ; 分配部　ｼﾌﾄ 動作異常
460   LD      T51  ; 分配部　着脱ﾌﾟｯｼｬｰ 動作異常
      OUT     B64  ; 分配部　着脱ﾌﾟｯｼｬｰ 動作異常
462   LD      T57  ; 着座つまり検知
      OUT     B65  ; 着座つまり検知
464   LD      T60  ; 締め部　ﾘﾀｰﾝｴｽｹｰﾌﾟ 動作異常
      OUT     B66  ; 締め部　ﾘﾀｰﾝｴｽｹｰﾌﾟ 動作異常
466   LD      T61  ; 締め部　ﾘﾀｰﾝｽﾄｯﾊﾟｰ 動作異常
      OUT     B67  ; 締め部　ﾘﾀｰﾝｽﾄｯﾊﾟｰ 動作異常
468   LD      T62  ; 締め部 ﾘﾌﾀｰ 動作異常
      OUT     B68  ; 締め部 ﾘﾌﾀｰ 動作異常
470   LD      T63  ; 締め部　着座確認　動作異常
      OUT     B69  ; 締め部　着座確認　動作異常
472   LD      T64  ; NGﾘﾌﾀｰ　動作異常
      OUT     B6A  ; NGﾘﾌﾀｰ　動作異常
474   LD      T65  ; 締め部　IDｾﾝｻｰ　動作異常
      OUT     B6B  ; 締め部　IDｾﾝｻｰ　動作異常
476   LD      T66  ; 締め部　ﾘﾌﾀｰ後　ｽﾄｯﾊﾟｰ　動作異常
      OUT     B6C  ; 締め部　ﾘﾌﾀｰ後　ｽﾄｯﾊﾟｰ　動作異常
478   LD      T67  ; 締め部　NRｽﾄｯﾊﾟｰ動作異常
      OUT     B6D  ; 締め部　NRｽﾄｯﾊﾟｰ動作異常
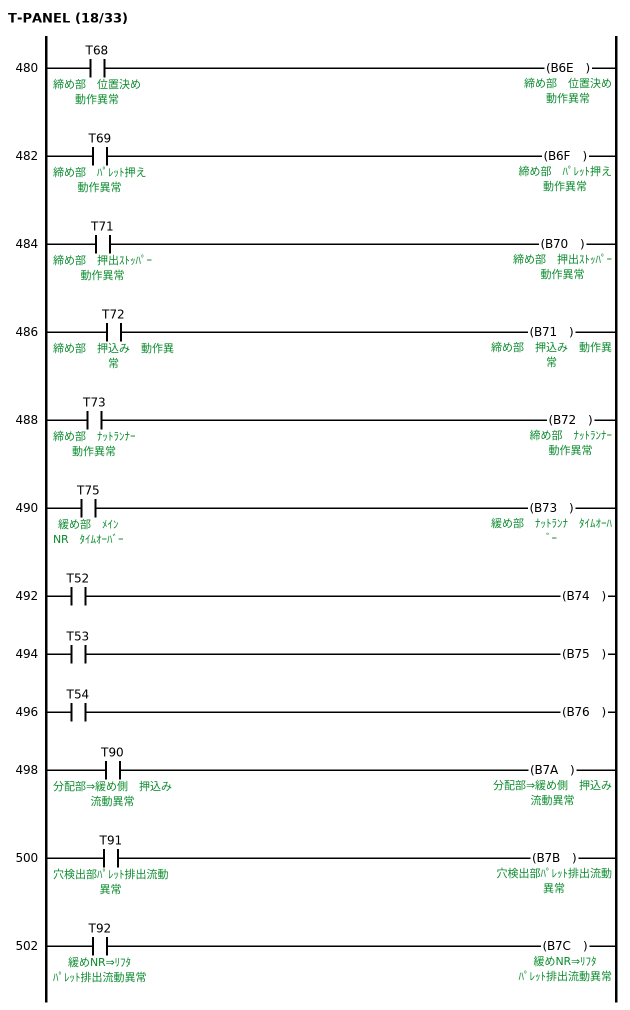
480   LD      T68  ; 締め部　位置決め 動作異常
      OUT     B6E  ; 締め部　位置決め 動作異常
482   LD      T69  ; 締め部　ﾊﾟﾚｯﾄ押え 動作異常
      OUT     B6F  ; 締め部　ﾊﾟﾚｯﾄ押え 動作異常
484   LD      T71  ; 締め部　押出ｽﾄｯﾊﾟｰ 動作異常
      OUT     B70  ; 締め部　押出ｽﾄｯﾊﾟｰ 動作異常
486   LD      T72  ; 締め部　押込み　動作異常
      OUT     B71  ; 締め部　押込み　動作異常
488   LD      T73  ; 締め部　ﾅｯﾄﾗﾝﾅｰ 動作異常
      OUT     B72  ; 締め部　ﾅｯﾄﾗﾝﾅｰ 動作異常
490   LD      T75  ; 緩め部　ﾒｲﾝ NR　ﾀｲﾑｵｰﾊﾞｰ
      OUT     B73  ; 緩め部　ﾅｯﾄﾗﾝﾅ　ﾀｲﾑｵｰﾊﾞｰ
492   LD      T52
      OUT     B74
494   LD      T53
      OUT     B75
496   LD      T54
      OUT     B76
498   LD      T90  ; 分配部⇒緩め側　押込み　流動異常
      OUT     B7A  ; 分配部⇒緩め側　押込み　流動異常
500   LD      T91  ; 穴検出部ﾊﾟﾚｯﾄ排出流動異常
      OUT     B7B  ; 穴検出部ﾊﾟﾚｯﾄ排出流動異常
502   LD      T92  ; 緩めNR⇒ﾘﾌﾀ ﾊﾟﾚｯﾄ排出流動異常
      OUT     B7C  ; 緩めNR⇒ﾘﾌﾀ ﾊﾟﾚｯﾄ排出流動異常
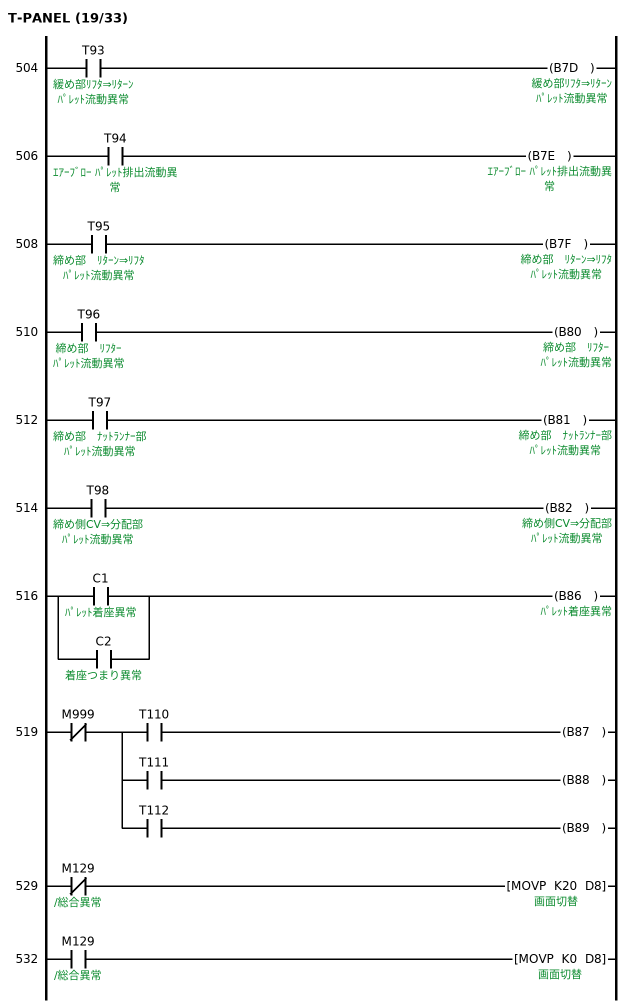
504   LD      T93  ; 緩め部ﾘﾌﾀ⇒ﾘﾀｰﾝ ﾊﾟﾚｯﾄ流動異常
      OUT     B7D  ; 緩め部ﾘﾌﾀ⇒ﾘﾀｰﾝ ﾊﾟﾚｯﾄ流動異常
506   LD      T94  ; ｴｱｰﾌﾞﾛｰ ﾊﾟﾚｯﾄ排出流動異常
      OUT     B7E  ; ｴｱｰﾌﾞﾛｰ ﾊﾟﾚｯﾄ排出流動異常
508   LD      T95  ; 締め部　ﾘﾀｰﾝ⇒ﾘﾌﾀ ﾊﾟﾚｯﾄ流動異常
      OUT     B7F  ; 締め部　ﾘﾀｰﾝ⇒ﾘﾌﾀ ﾊﾟﾚｯﾄ流動異常
510   LD      T96  ; 締め部　ﾘﾌﾀｰ ﾊﾟﾚｯﾄ流動異常
      OUT     B80  ; 締め部　ﾘﾌﾀｰ ﾊﾟﾚｯﾄ流動異常
512   LD      T97  ; 締め部　ﾅｯﾄﾗﾝﾅｰ部 ﾊﾟﾚｯﾄ流動異常
      OUT     B81  ; 締め部　ﾅｯﾄﾗﾝﾅｰ部 ﾊﾟﾚｯﾄ流動異常
514   LD      T98  ; 締め側CV⇒分配部 ﾊﾟﾚｯﾄ流動異常
      OUT     B82  ; 締め側CV⇒分配部 ﾊﾟﾚｯﾄ流動異常
516   LD      C1  ; ﾊﾟﾚｯﾄ着座異常
      OR      C2  ; 着座つまり異常
      OUT     B86  ; ﾊﾟﾚｯﾄ着座異常
519   LDI     M999
      MPS
      AND     T110
      OUT     B87
      MRD
      AND     T111
      OUT     B88
      MPP
      AND     T112
      OUT     B89
529   LDI     M129  ; /総合異常
      MOVP    K20 D8  ; 画面切替
532   LD      M129  ; /総合異常
      MOVP    K0 D8
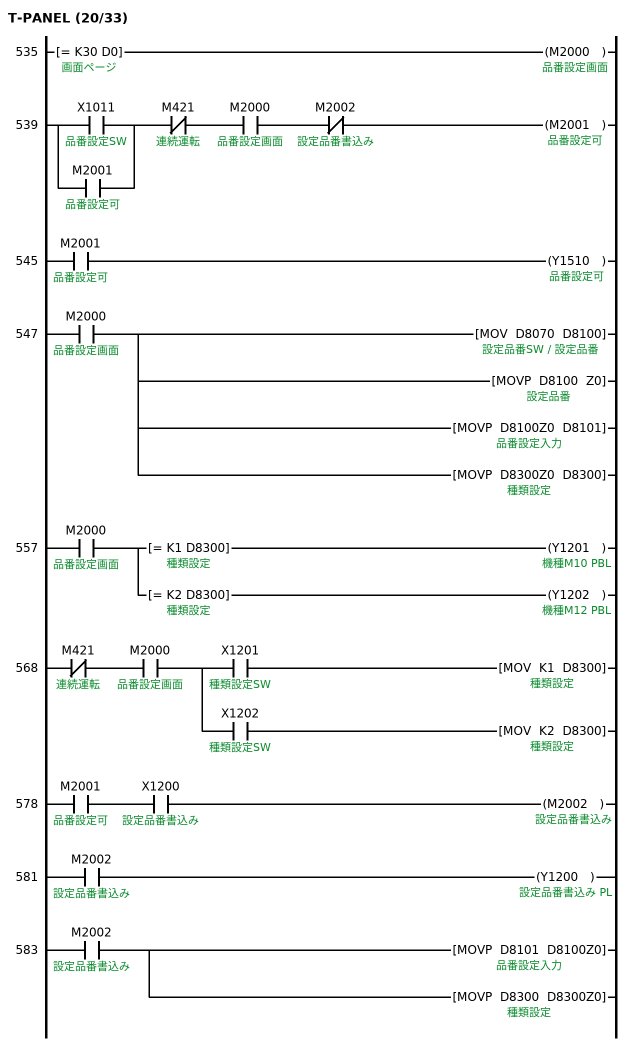
535   LD=     K30 D0  ; 画面ページ
      OUT     M2000  ; 品番設定画面
539   LD      X1011  ; 品番設定SW
      OR      M2001  ; 品番設定可
      ANI     M421  ; 連続運転
      AND     M2000  ; 品番設定画面
      ANI     M2002  ; 設定品番書込み
      OUT     M2001  ; 品番設定可
545   LD      M2001  ; 品番設定可
      OUT     Y1510  ; 品番設定可
547   LD      M2000  ; 品番設定画面
      MOV     D8070 D8100  ; 設定品番SW / 設定品番
      MOVP    D8100 Z0
      MOVP    D8100Z0 D8101  ; 品番設定入力
      MOVP    D8300Z0 D8300  ; 種類設定
557   LD      M2000  ; 品番設定画面
      MPS
      AND=    K1 D8300  ; 種類設定
      OUT     Y1201  ; 機種M10 PBL
      MPP
      AND=    K2 D8300  ; 種類設定
      OUT     Y1202  ; 機種M12 PBL
568   LDI     M421  ; 連続運転
      AND     M2000  ; 品番設定画面
      MPS
      AND     X1201  ; 種類設定SW
      MOV     K1 D8300
      MPP
      AND     X1202  ; 種類設定SW
      MOV     K2 D8300
578   LD      M2001  ; 品番設定可
      AND     X1200  ; 設定品番書込み
      OUT     M2002  ; 設定品番書込み
581   LD      M2002  ; 設定品番書込み
      OUT     Y1200  ; 設定品番書込み PL
583   LD      M2002  ; 設定品番書込み
      MOVP    D8101 D8100Z0
      MOVP    D8300 D8300Z0
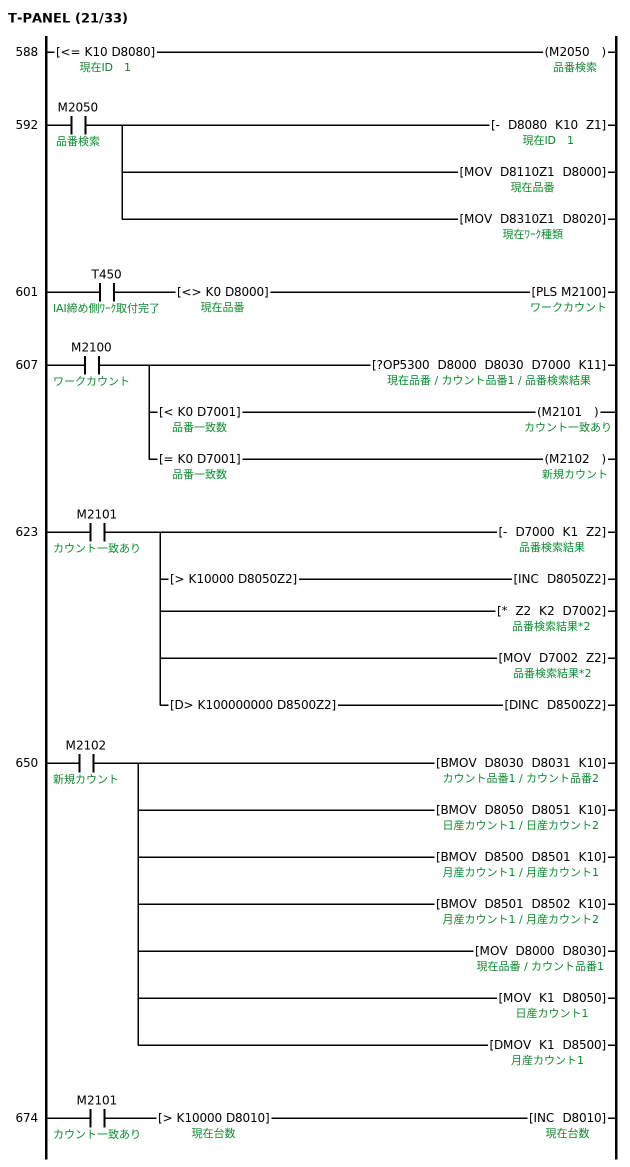
588   LD<=    K10 D8080  ; 現在ID　1
      OUT     M2050  ; 品番検索
592   LD      M2050  ; 品番検索
      -       D8080 K10 Z1
      MOV     D8110Z1 D8000  ; 現在品番
      MOV     D8310Z1 D8020  ; 現在ﾜｰｸ種類
601   LD      T450  ; IAI締め側ﾜｰｸ取付完了
      AND<>   K0 D8000  ; 現在品番
      PLS     M2100  ; ワークカウント
607   LD      M2100  ; ワークカウント
      ?OP5300 D8000 D8030 D7000 K11  ; カウント品番1 / 品番検索結果
      MPS
      AND<    K0 D7001  ; 品番一致数
      OUT     M2101  ; カウント一致あり
      MPP
      AND=    K0 D7001  ; 品番一致数
      OUT     M2102  ; 新規カウント
623   LD      M2101  ; カウント一致あり
      -       D7000 K1 Z2
      MPS
      AND>    K10000 D8050Z2
      INC     D8050Z2
      MPP
      *       Z2 K2 D7002  ; 品番検索結果*2
      MOV     D7002 Z2
      ANDD>   K100000000 D8500Z2
      DINC    D8500Z2
650   LD      M2102  ; 新規カウント
      BMOV    D8030 D8031 K10  ; カウント品番2
      BMOV    D8050 D8051 K10  ; 日産カウント1 / 日産カウント2
      BMOV    D8500 D8501 K10  ; 月産カウント1 / 月産カウント1
      BMOV    D8501 D8502 K10  ; 月産カウント2
      MOV     D8000 D8030
      MOV     K1 D8050
      DMOV    K1 D8500
674   LD      M2101  ; カウント一致あり
      AND>    K10000 D8010  ; 現在台数
      INC     D8010
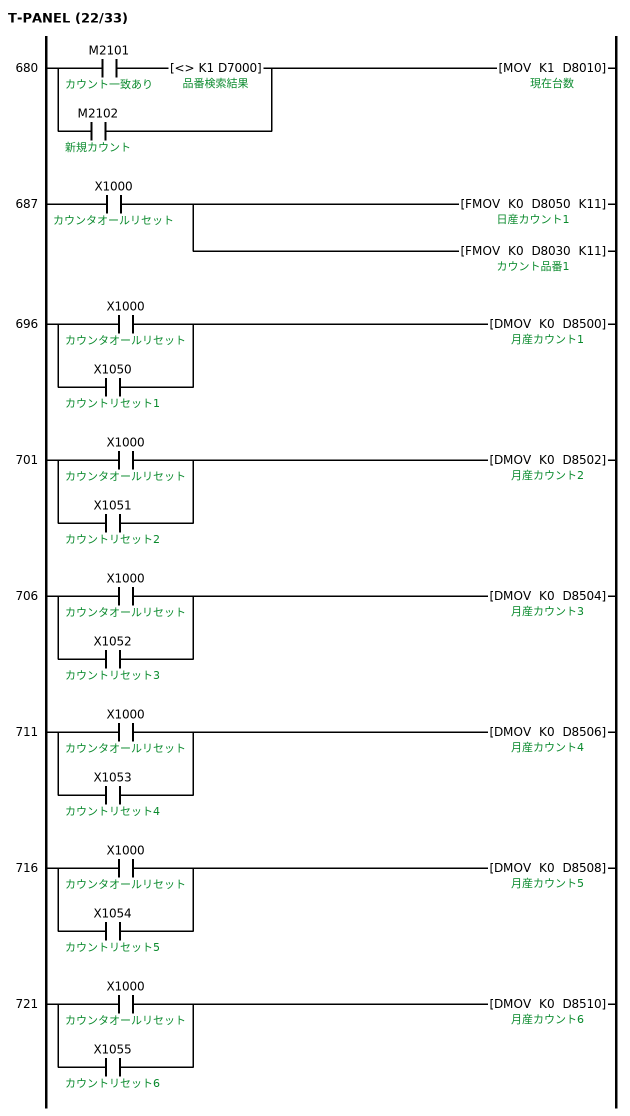
680   LD      M2101  ; カウント一致あり
      AND<>   K1 D7000  ; 品番検索結果
      OR      M2102  ; 新規カウント
      MOV     K1 D8010
687   LD      X1000  ; カウンタオールリセット
      FMOV    K0 D8050 K11
      FMOV    K0 D8030 K11
696   LD      X1000  ; カウンタオールリセット
      OR      X1050  ; カウントリセット1
      DMOV    K0 D8500
701   LD      X1000  ; カウンタオールリセット
      OR      X1051  ; カウントリセット2
      DMOV    K0 D8502
706   LD      X1000  ; カウンタオールリセット
      OR      X1052  ; カウントリセット3
      DMOV    K0 D8504  ; 月産カウント3
711   LD      X1000  ; カウンタオールリセット
      OR      X1053  ; カウントリセット4
      DMOV    K0 D8506  ; 月産カウント4
716   LD      X1000  ; カウンタオールリセット
      OR      X1054  ; カウントリセット5
      DMOV    K0 D8508  ; 月産カウント5
721   LD      X1000  ; カウンタオールリセット
      OR      X1055  ; カウントリセット6
      DMOV    K0 D8510  ; 月産カウント6
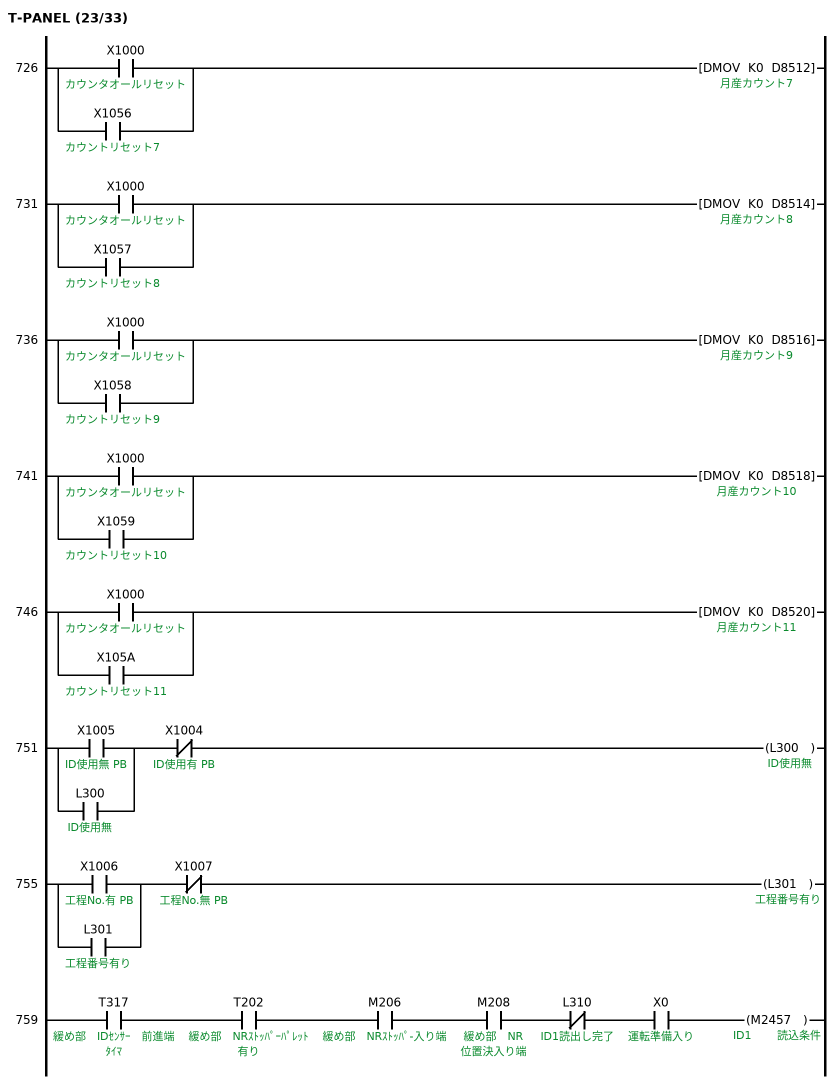
726   LD      X1000  ; カウンタオールリセット
      OR      X1056  ; カウントリセット7
      DMOV    K0 D8512  ; 月産カウント7
731   LD      X1000  ; カウンタオールリセット
      OR      X1057  ; カウントリセット8
      DMOV    K0 D8514  ; 月産カウント8
736   LD      X1000  ; カウンタオールリセット
      OR      X1058  ; カウントリセット9
      DMOV    K0 D8516  ; 月産カウント9
741   LD      X1000  ; カウンタオールリセット
      OR      X1059  ; カウントリセット10
      DMOV    K0 D8518  ; 月産カウント10
746   LD      X1000  ; カウンタオールリセット
      OR      X105A  ; カウントリセット11
      DMOV    K0 D8520  ; 月産カウント11
751   LD      X1005  ; ID使用無 PB
      OR      L300  ; ID使用無
      ANI     X1004  ; ID使用有 PB
      OUT     L300  ; ID使用無
755   LD      X1006  ; 工程No.有 PB
      OR      L301  ; 工程番号有り
      ANI     X1007  ; 工程No.無 PB
      OUT     L301  ; 工程番号有り
759   LD      T317  ; 緩め部　IDｾﾝｻｰ　前進端ﾀｲﾏ
      AND     T202  ; 緩め部　NRｽﾄｯﾊﾟｰﾊﾟﾚｯﾄ有り
      AND     M206  ; 緩め部　NRｽﾄｯﾊﾟ-入り端
      AND     M208  ; 緩め部　NR 位置決入り端
      ANI     L310  ; ID1読出し完了
      AND     X0  ; 運転準備入り
      OUT     M2457  ; ID1 　　読込条件
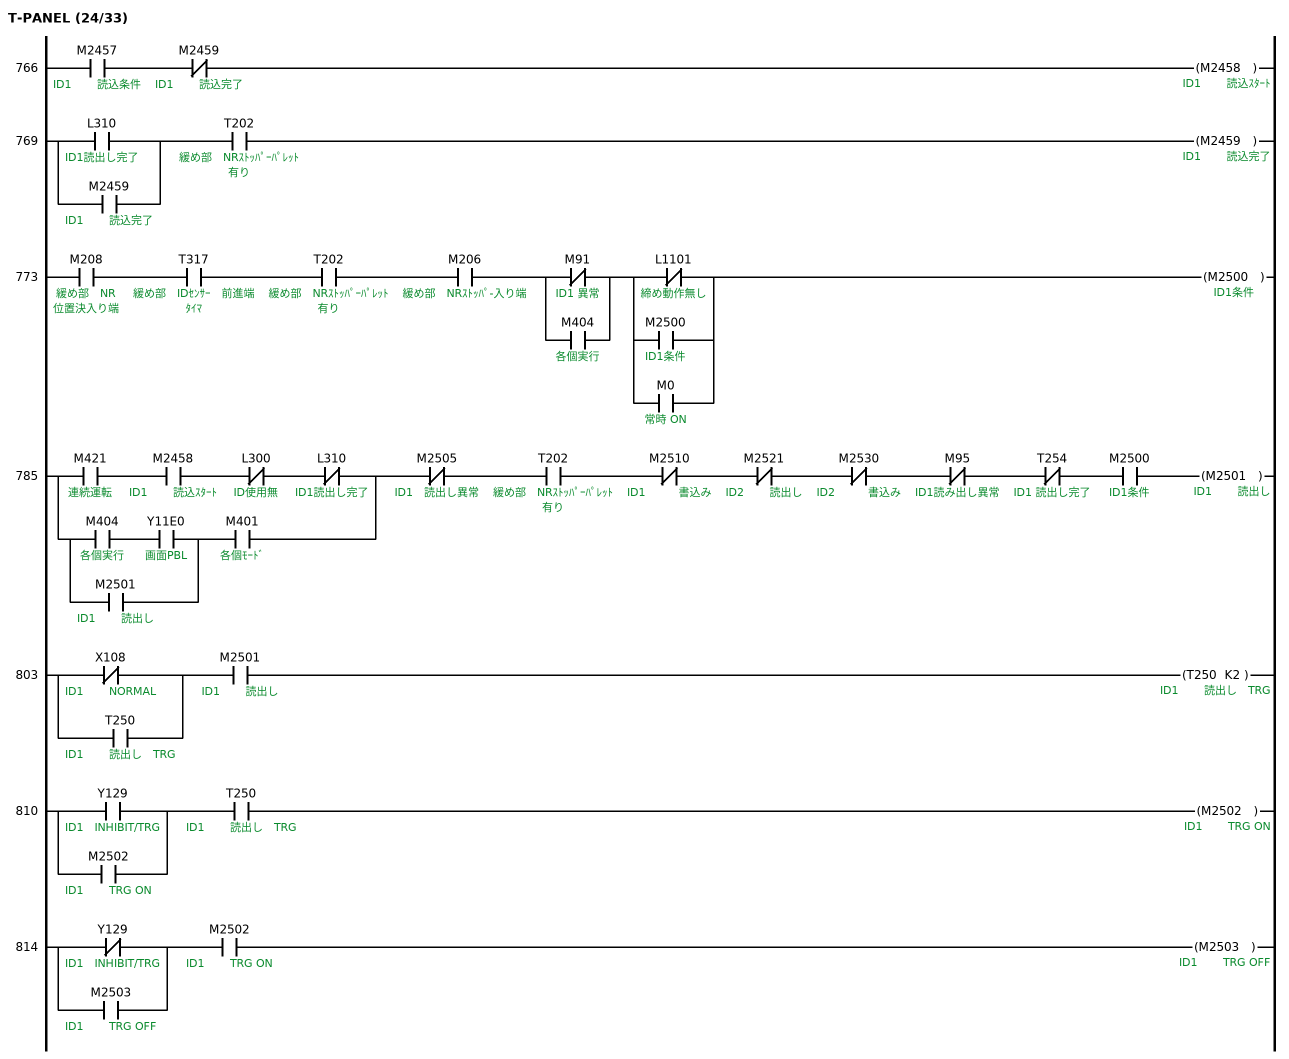
766   LD      M2457  ; ID1 　　読込条件
      ANI     M2459  ; ID1 　　読込完了
      OUT     M2458  ; ID1 　　読込ｽﾀｰﾄ
769   LD      L310  ; ID1読出し完了
      OR      M2459  ; ID1 　　読込完了
      AND     T202  ; 緩め部　NRｽﾄｯﾊﾟｰﾊﾟﾚｯﾄ有り
      OUT     M2459  ; ID1 　　読込完了
773   LD      M208  ; 緩め部　NR 位置決入り端
      AND     T317  ; 緩め部　IDｾﾝｻｰ　前進端ﾀｲﾏ
      AND     T202  ; 緩め部　NRｽﾄｯﾊﾟｰﾊﾟﾚｯﾄ有り
      AND     M206  ; 緩め部　NRｽﾄｯﾊﾟ-入り端
      LDI     M91  ; ID1 異常
      OR      M404  ; 各個実行
      ANB
      LDI     L1101  ; 締め動作無し
      OR      M2500  ; ID1条件
      OR      M0  ; 常時 ON
      ANB
      OUT     M2500  ; ID1条件
785   LD      M421  ; 連続運転
      AND     M2458  ; ID1 　　読込ｽﾀｰﾄ
      ANI     L300  ; ID使用無
      ANI     L310  ; ID1読出し完了
      LD      M404  ; 各個実行
      AND     Y11E0  ; 画面PBL
      OR      M2501  ; ID1　 　読出し
      AND     M401  ; 各個ﾓｰﾄﾞ
      ORB
      ANI     M2505  ; ID1　読出し異常
      AND     T202  ; 緩め部　NRｽﾄｯﾊﾟｰﾊﾟﾚｯﾄ有り
      ANI     M2510  ; ID1　　　書込み
      ANI     M2521  ; ID2　 　読出し
      ANI     M2530  ; ID2　　　書込み
      ANI     M95  ; ID1読み出し異常
      ANI     T254  ; ID1 読出し完了
      AND     M2500  ; ID1条件
      OUT     M2501  ; ID1　 　読出し
803   LDI     X108  ; ID1　　 NORMAL
      OR      T250  ; ID1　 　読出し　TRG
      AND     M2501  ; ID1　 　読出し
      OUT     T250 K2  ; ID1　 　読出し　TRG
810   LD      Y129  ; ID1　INHIBIT/TRG
      OR      M2502  ; ID1　 　TRG ON
      AND     T250  ; ID1　 　読出し　TRG
      OUT     M2502  ; ID1　 　TRG ON
814   LDI     Y129  ; ID1　INHIBIT/TRG
      OR      M2503  ; ID1　 　TRG OFF
      AND     M2502  ; ID1　 　TRG ON
      OUT     M2503  ; ID1　 　TRG OFF
